{attribute addProperty BoxType "EL6688-0000-0022"}
{attribute addProperty Id "External_SyncAT %I*External_Sync_07348351192240WcStateAT %I*WcState_98A4DF7520.250InfoDataAT %I*InfoData_0BDED7BF144180"}
{attribute addProperty CRC "701044449"}
{attribute addProperty SizeInBites "338"}
{attribute addProperty SizeInBytes "42.25"}
TYPE EL6688_092E4D1F :
STRUCT
	{attribute addProperty Name "External_Sync"}
	External_Sync : External_Sync_07348351;
	{attribute addProperty Name "WcState"}
	WcState : WcState_98A4DF75;
	{attribute addProperty Name "InfoData"}
	InfoData : InfoData_0BDED7BF;
END_STRUCT
END_TYPE

(* stored: Version 1.2.0.0, ProductVersion 3.1.4024.9
   DUT EL6688_092E4D1F: Id {12c0563c-48a3-4b51-a656-f4aa731d696a} *)
